// TwinCAT 3 PLC project Untitled1
// ProgramVersion: 3.1.4023.0
// libraries:
//   Tc2_Standard, * (Beckhoff Automation GmbH)
//   Tc2_System, * (Beckhoff Automation GmbH)
//   Tc3_Module, * (Beckhoff Automation GmbH)
// project tree:
//   DUTs/ DataDrill.TcDUT, INPUT.TcDUT, OUTPUT.TcDUT
//   / GlobalTextList.TcGTLO, PlcTask.TcTTO, Visualization Manager.TcVMO (not stored)
//   POUs/ MAIN.TcPOU
//   VISUs/ Visualization.TcVIS
// real-time tasks:
//   TASK PlcTask: cycle T#10ms, priority 20, ADS port 350

CONFIGURATION Untitled1
    RESOURCE PLC ON TwinCAT3
        TASK PlcTask(INTERVAL := T#10ms, PRIORITY := 20);
        PROGRAM MAIN WITH PlcTask : MAIN;
    END_RESOURCE
END_CONFIGURATION

// ---- DUTs/DataDrill.TcDUT
TYPE DataDrill :
STRUCT
	
	OUT	:	OUTPUT;
	IN	:	INPUT;

END_STRUCT
END_TYPE

// ---- DUTs/INPUT.TcDUT
TYPE INPUT :
STRUCT
	

	bStart 		:	BOOL;	//S1 Butonu , NO
	
	bUpSwitch 	:	BOOL;	//ÜÖN , NC
	
	bSwitchA	:	BOOL;	// A anahtarı, NO
	bSwitchB	:	BOOL;	// B anahtarı , NC
	bSwitchC	:	BOOL;	// C anahtarı , NO
	
	


END_STRUCT
END_TYPE

// ---- DUTs/OUTPUT.TcDUT
TYPE OUTPUT :
STRUCT
	
	bDrill	:	BOOL;	//Matkap M1
	bUp		:	BOOL;	// Yukarı Komutu
	bDown	:	BOOL;	//Aşağı Komutu

END_STRUCT
END_TYPE

// ---- POUs/MAIN.TcPOU
PROGRAM MAIN
VAR
	
	Drill	:	DataDrill;
	Drill2	:	DataDrill;

	nState: INT;
	ftrigA: F_TRIG;
	
	rtrigA: R_TRIG;
	
	ftrigB: F_TRIG;
	ftrigUON: F_TRIG;
	
	fDrillY: REAL;
	C: BOOL;
END_VAR


C	:=	NOT(Drill.IN.bSwitchC);

ACT_MatkapUygulamasi();
ACT_Visu();

ACTION ACT_MatkapUygulamasi:

rtrigA(CLK:= Drill.IN.bSwitchA , Q=> );
ftrigA(CLK:= Drill.IN.bSwitchA , Q=> );


ftrigB(CLK:= Drill.IN.bSwitchB , Q=> );
ftrigUON(CLK:= Drill.IN.bUpSwitch , Q=> );



CASE nState OF
	

	0:
	
		Drill.OUT.bDown	:=	FALSE;
		Drill.OUT.bUp	:=	FALSE;
	
		IF Drill.IN.bStart AND 
		NOT Drill.IN.bUpSwitch AND
		 Drill.IN.bSwitchC	THEN
		 
			nState := 10;
		
		END_IF
	
		
	10:
		
		Drill.OUT.bDown	:=	TRUE;
		
		IF rtrigA.Q AND Drill.IN.bSwitchC THEN
			
			nState := 20;
			
		ELSIF NOT Drill.IN.bSwitchC THEN
			
			nState := 999;
			
		END_IF
	
		
	20:	
	
		Drill.OUT.bDrill	:=	TRUE;
		
		
		IF ftrigB.Q AND Drill.IN.bSwitchC THEN
			
			nState := 30;
			
		ELSIF NOT Drill.IN.bSwitchC THEN
			
			nState := 999;
			
		END_IF	
	
	30:
	
		Drill.OUT.bDown	:=	FALSE;
		Drill.OUT.bUp	:=	TRUE;
	
		IF ftrigA.Q  AND Drill.IN.bSwitchC THEN 

			nState := 40;
			
		ELSIF NOT Drill.IN.bSwitchC THEN
		
			nState := 999;
			
		END_IF
		
	40:
	
		Drill.OUT.bDrill	:=	FALSE;

		IF ftrigUON.Q THEN
			
		Drill.OUT.bDown	:=	FALSE;
		Drill.OUT.bUp	:=	FALSE;
		
			nState := 0;
			
		END_IF
	

END_CASE



	IF NOT Drill.IN.bStart	THEN  
			 
		nState := 0;
		Drill.OUT.bDown	:=	FALSE;
		Drill.OUT.bUp	:=	FALSE;		
		Drill.OUT.bDrill	:=	FALSE;
	
	END_IF
END_ACTION

ACTION ACT_Visu:


//50-225

IF Drill.OUT.bDown AND NOT Drill.OUT.bUp THEN
	
	fDrillY	:=	fDrillY + 0.5;
	
	IF fDrillY	>=	100 AND NOT Drill.OUT.bDrill THEN
		fDrillY	:=	100;
	
	
	ELSIF Drill.OUT.bDrill THEN
	
		fDrillY	:=	fDrillY + 0.3;
		
	IF fDrillY	>=	200	THEN
		
		fDrillY	:=	200;
		
	END_IF
	
	END_IF
	

	
ELSIF Drill.OUT.bUp AND NOT Drill.OUT.bDown AND Drill.OUT.bDrill THEN
	
	fDrillY	:=	fDrillY	-	0.3;
	
	IF fDrillY	<=	50	THEN
		fDrillY	:=	50;
	END_IF	

ELSIF Drill.OUT.bUp AND NOT Drill.OUT.bDown AND NOT Drill.OUT.bDrill THEN
	
	fDrillY	:=	fDrillY	-	0.5;
	
	IF fDrillY	<=	20	THEN
		
		fDrillY	:=	20;
		
	END_IF	
	
	
END_IF
END_ACTION

END_PROGRAM

// ---- GlobalTextList.TcGTLO
TEXTLIST GlobalTextList
  437 = 'Aşağı'
  377 = 'GroupBox'
  409 = 'Label'
  10 = 'Matkap'
  979 = 'Sistem Durumu'
  987 = 'Sistem Kontrol'
  517 = 'SwitchA'
  105 = 'SwitchB'
  827 = 'SwitchC'
  485 = 'Yukarı'
  173 = 'ÜÖN'
END_TEXTLIST

// ---- VISUs/Visualization.TcVIS
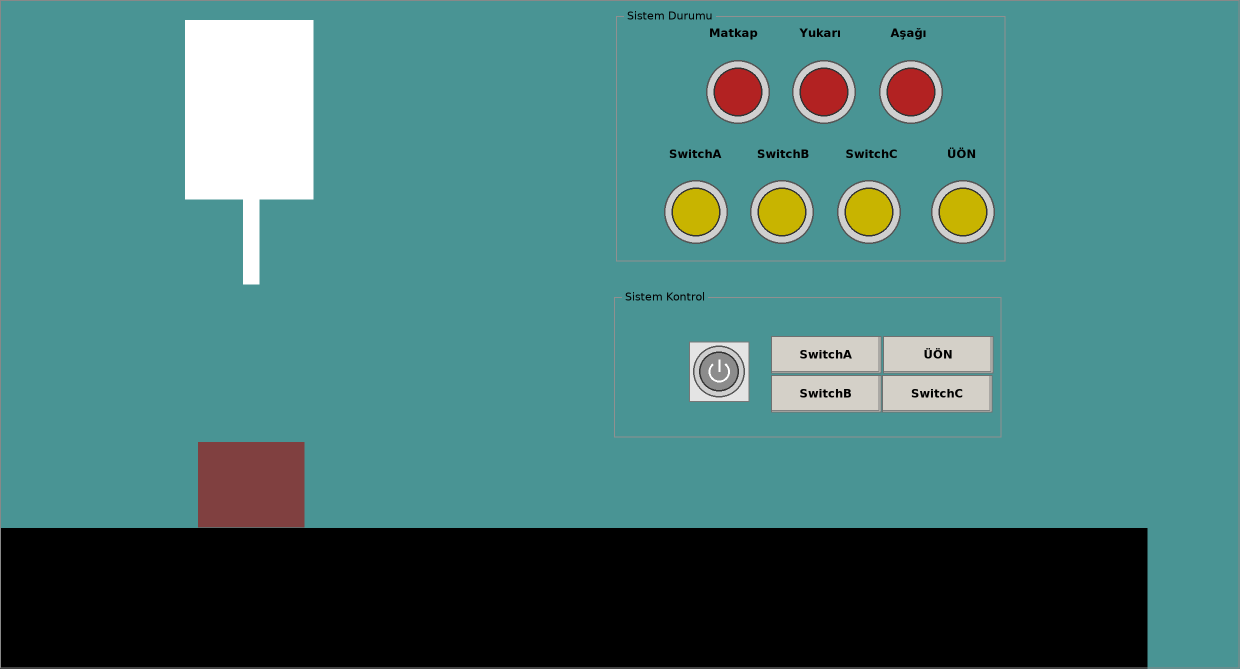
VISUALIZATION Visualization  // 1240x669
    Rectangle (-93,528 1240x141)
    Rectangle (198,442 106x85), invisible if: MAIN.C
    Group (185,20 128x264)
        p2738717112: MAIN.fDrillY
        Rectangle (58,164 16x100)
        Rectangle (0,0 128x179)
    Lamp1 (699,55 78x74), variable: MAIN.Drill.OUT.bDrill, style: Lamp-Lamp1-Red
    Lamp1 (785,55 78x74), variable: MAIN.Drill.OUT.bUp, style: Lamp-Lamp1-Red
    Lamp1 (872,55 78x74), variable: MAIN.Drill.OUT.bDown, style: Lamp-Lamp1-Red
    Label (702,18 63x30), "Matkap"
    Label (789,18 63x30), "Yukarı"
    Label (877,18 63x30), "Aşağı"
    Lamp1 (657,175 78x74), variable: MAIN.Drill.IN.bSwitchA, style: Lamp-Lamp1-Yellow
    Lamp1 (743,175 78x74), variable: MAIN.Drill.IN.bSwitchB, style: Lamp-Lamp1-Yellow
    Lamp1 (830,175 78x74), variable: MAIN.Drill.IN.bSwitchC, style: Lamp-Lamp1-Yellow
    Lamp1 (924,175 78x74), variable: MAIN.Drill.IN.bUpSwitch, style: Lamp-Lamp1-Yellow
    Label (664,139 63x30), "SwitchA"
    Label (752,139 63x30), "SwitchB"
    Label (840,139 63x30), "SwitchC"
    Label (930,139 63x30), "ÜÖN"
    Button (771,336 110x37), "SwitchA"
        toggle MAIN.Drill.IN.bSwitchA
    Button (771,375 110x37), "SwitchB"
        toggle MAIN.Drill.IN.bSwitchB
    Button (882,375 110x37), "SwitchC"
        toggle MAIN.Drill.IN.bSwitchC
    Button (883,336 110x37), "ÜÖN"
        toggle MAIN.Drill.IN.bUpSwitch
    PowerSwitch (689,341 60x61), variable: MAIN.Drill.IN.bStart, behaviour: TOGGLE, style: Switch-PowerSwitch-Gray
    GroupBox (616,8 389x253), "Sistem Durumu"
    GroupBox (614,289 387x148), "Sistem Kontrol"
END_VISUALIZATION
